// TIA Portal project "2022.06.08_FC的应用" (V17)

(* hardware
DEVICE "S7-1200 station_1"  S7-1200 Station
   slot 0: "Rack_0"  S7-1200 Rack  Rack  V1.0
   slot 1: "PLC_1"  CPU 1212C DC/DC/DC  6ES7 212-1AE40-0XB0  V4.5
*)

// ===== PLC "PLC_1"  CPU 1212C DC/DC/DC =====

VAR_GLOBAL   // PLC tag table "默认变量表"
   "模拟量输入" AT %MW100 : Word;
   "Tag_3" AT %MW102 : UInt;
   "Tag_4" AT %MW104 : UInt;
   "Tag_5" AT %MW106 : UInt;
   "Tag_6" AT %I0.0 : Bool;
   "Tag_7" AT %M0.0 : Bool;
   "X(2)" AT %MW10 : Word;
   "Tag_9" AT %MW12 : UInt;
   "X" AT %MW0 : Word;
   "a" AT %MW2 : Word;
   "b" AT %MW4 : Int;
   "c" AT %MW8 : Int;
   "实时温度" AT %MD0 : Real;
   "Tag_10" AT %MD2 : Real;
   "f" AT %MD4 : Real;
   "g" AT %MD8 : Real;
   "X(1)" AT %MD12 : Real;
   "Tag_8" AT %MD16 : Real;
   "中间值(1)" AT %MD200 : Real;
   "中间值" AT %MD104 : Real;
   "工程值" AT %MD108 : Real;
   "要求的频率" AT %MD60 : Real;
   "百分比" AT %MD64 : Real;
   "Tag_12" AT %MW70 : Int;
   "Tag_2" AT %I0.1 : Bool;
   "0" AT %Q0.0 : Bool;
   "加热" AT %Q0.1 : Bool;
   "Tag_1" AT %MD100 : Time;
   "Tag_11" AT %M0.1 : Bool;
   "Tag_13" AT %QB0 : Byte;
   "Tag_14" AT %QB1 : Byte;
   "Tag_15" AT %M0.2 : Bool;
   "Tag_16" AT %QB2 : Byte;
   "Tag_17" AT %I0.2 : Bool;
   "Tag_18" AT %M10.0 : Bool;
   "Tag_19" AT %Q0.2 : Bool;
   "Tag_20" AT %I0.3 : Bool;
END_VAR

DATA_BLOCK "测试数据块_1"   // DB1
{ S7_Optimized_Access := 'FALSE' }
VERSION : 0.1
BEGIN
END_DATA_BLOCK

FUNCTION "起保停" : Void   // FC1, LAD
{ S7_Optimized_Access := 'TRUE' }
VERSION : 0.1
BEGIN

REGION Network 1
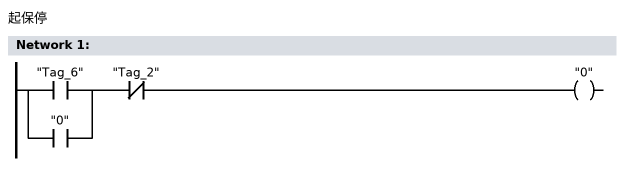
   RUNG wire#powerrail
      Contact( "Tag_6" )
      wire#w1
      I_Contact( "Tag_2" )
      Coil( "0" )
   END_RUNG
   RUNG wire#powerrail
      Contact( "0" )
   END_RUNG wire#w1
   // the same network as SCL:
   "0" := ("Tag_6" OR "0") AND NOT "Tag_2";
END_REGION
END_FUNCTION

FUNCTION "正反转" : Void   // FC2, LAD
{ S7_Optimized_Access := 'TRUE' }
VERSION : 0.1
BEGIN

REGION Network 1
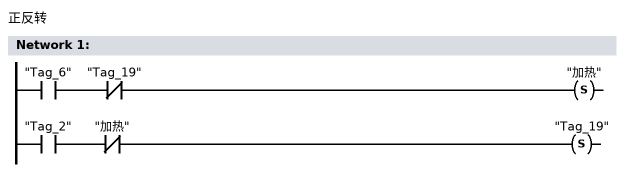
   RUNG wire#powerrail
      Contact( "Tag_6" )
      I_Contact( "Tag_19" )
      S_Coil( "加热" )
   END_RUNG
   RUNG wire#powerrail
      Contact( "Tag_2" )
      I_Contact( "加热" )
      S_Coil( "Tag_19" )
   END_RUNG
   // the same network as SCL:
   IF "Tag_6" AND NOT "Tag_19" THEN "加热" := TRUE; END_IF;
   IF "Tag_2" AND NOT "加热" THEN "Tag_19" := TRUE; END_IF;
END_REGION
END_FUNCTION

ORGANIZATION_BLOCK "Main"   // OB1, LAD, ProgramCycle
TITLE = "Main Program Sweep (Cycle)"
{ S7_Optimized_Access := 'TRUE' }
VERSION : 0.1
   VAR_INPUT
      Initial_Call : Bool;   // Initial call of this OB
      Remanence : Bool;   // =True, if remanent data are available
   END_VAR
BEGIN

REGION Network 1
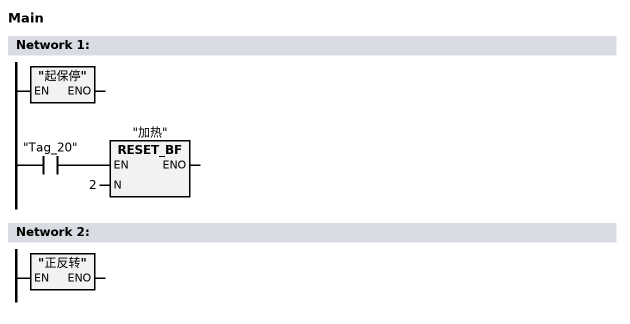
   // no SCL statement known for RBitfield: written as a call
   "起保停"();
   IF "Tag_20" THEN RESET_BF(operand := "加热", n := 2); END_IF;
END_REGION

REGION Network 2
   RUNG wire#powerrail
      "正反转"()
   END_RUNG
   // the same network as SCL:
   "正反转"();
END_REGION
END_ORGANIZATION_BLOCK